// TIA Portal V16 export
// export: Created 2024-05-10T06:46:45.280441Z, ExportSetting WithDefaults, DisplayName Totally Integrated Automation Portal, DisplayVersion V16, DisplayName TIA Portal Version Control Interface, DisplayVersion V16, DisplayName TIA Portal Openness, DisplayVersion V16, DisplayName STEP 7 Professional, DisplayVersion V16, DisplayName STEP 7 Safety, DisplayVersion V16, DisplayName WinCC Professional, DisplayVersion V16
VAR_GLOBAL   // PLC tag table "105阀控制变量表"
   EN_阻挡下指令自动 AT %M2000.0 : Bool;
   EN_阻挡上指令自动 AT %M2000.1 : Bool;
   EN_提升机下指令自动 AT %M2000.4 : Bool;
   EN_提升机上指令自动 AT %M2000.5 : Bool;
   EX_阻挡下指令自动 AT %M2001.0 : Bool;
   EX_阻挡上指令自动 AT %M2001.1 : Bool;
   EX_提升机下指令自动 AT %M2001.4 : Bool;
   EX_提升机上指令自动 AT %M2001.5 : Bool;
   ST01上阻挡下指令自动 AT %M2002.0 : Bool;
   ST01上阻挡上指令自动 AT %M2002.1 : Bool;
   ST01下阻挡下指令自动 AT %M2002.4 : Bool;
   ST01下阻挡上指令自动 AT %M2002.5 : Bool;
   ST02上阻挡下指令自动 AT %M2003.0 : Bool;
   ST02上阻挡上指令自动 AT %M2003.1 : Bool;
   ST02下阻挡下指令自动 AT %M2003.4 : Bool;
   ST02下阻挡上指令自动 AT %M2003.5 : Bool;
   ST03上阻挡下指令自动 AT %M2004.0 : Bool;
   ST03上阻挡上指令自动 AT %M2004.1 : Bool;
   ST03下阻挡下指令自动 AT %M2004.4 : Bool;
   ST03下阻挡上指令自动 AT %M2004.5 : Bool;
   ST04上阻挡下指令自动 AT %M2005.0 : Bool;
   ST04上阻挡上指令自动 AT %M2005.1 : Bool;
   ST05上阻挡下指令自动 AT %M2005.4 : Bool;
   ST05上阻挡上指令自动 AT %M2005.5 : Bool;
   ST06上阻挡下指令自动 AT %M2006.0 : Bool;
   ST06上阻挡上指令自动 AT %M2006.1 : Bool;
   ST07上阻挡下指令自动 AT %M2006.4 : Bool;
   ST07上阻挡上指令自动 AT %M2006.5 : Bool;
   ST08上阻挡下指令自动 AT %M2007.0 : Bool;
   ST08上阻挡上指令自动 AT %M2007.1 : Bool;
   ST09上阻挡下指令自动 AT %M2007.4 : Bool;
   ST09上阻挡上指令自动 AT %M2007.5 : Bool;
   ST10上阻挡下指令自动 AT %M2008.0 : Bool;
   ST10上阻挡上指令自动 AT %M2008.1 : Bool;
   ST11上阻挡下指令自动 AT %M2008.4 : Bool;
   ST11上阻挡上指令自动 AT %M2008.5 : Bool;
   ST12上阻挡下指令自动 AT %M2009.0 : Bool;
   ST12上阻挡上指令自动 AT %M2009.1 : Bool;
   阀20进指令自动 AT %M2009.4 : Bool;
   阀20回指令自动 AT %M2009.5 : Bool;
   阀21进指令自动 AT %M2010.0 : Bool;
   阀21回指令自动 AT %M2010.1 : Bool;
   阀22进指令自动 AT %M2010.4 : Bool;
   阀22回指令自动 AT %M2010.5 : Bool;
   阀23进指令自动 AT %M2011.0 : Bool;
   阀23回指令自动 AT %M2011.1 : Bool;
   阀24进指令自动 AT %M2011.4 : Bool;
   阀24回指令自动 AT %M2011.5 : Bool;
   阀25进指令自动 AT %M2012.0 : Bool;
   阀25回指令自动 AT %M2012.1 : Bool;
   阀26进指令自动 AT %M2012.4 : Bool;
   阀26回指令自动 AT %M2012.5 : Bool;
   阀27进指令自动 AT %M2013.0 : Bool;
   阀27回指令自动 AT %M2013.1 : Bool;
   阀28进指令自动 AT %M2013.4 : Bool;
   阀28回指令自动 AT %M2013.5 : Bool;
   阀29进指令自动 AT %M2014.0 : Bool;
   阀29回指令自动 AT %M2014.1 : Bool;
   阀30进指令自动 AT %M2014.4 : Bool;
   阀30回指令自动 AT %M2014.5 : Bool;
   阀31进指令自动 AT %M2015.0 : Bool;
   阀31回指令自动 AT %M2015.1 : Bool;
   阀32进指令自动 AT %M2015.4 : Bool;
   阀32回指令自动 AT %M2015.5 : Bool;
   阀33进指令自动 AT %M2016.0 : Bool;
   阀33回指令自动 AT %M2016.1 : Bool;
   阀34进指令自动 AT %M2016.4 : Bool;
   阀34回指令自动 AT %M2016.5 : Bool;
   阀35进指令自动 AT %M2017.0 : Bool;
   阀35回指令自动 AT %M2017.1 : Bool;
   阀36进指令自动 AT %M2017.4 : Bool;
   阀36回指令自动 AT %M2017.5 : Bool;
   阀37进指令自动 AT %M2018.0 : Bool;
   阀37回指令自动 AT %M2018.1 : Bool;
   阀38进指令自动 AT %M2018.4 : Bool;
   阀38回指令自动 AT %M2018.5 : Bool;
   阀39进指令自动 AT %M2019.0 : Bool;
   阀39回指令自动 AT %M2019.1 : Bool;
   阀40进指令自动 AT %M2019.4 : Bool;
   阀40回指令自动 AT %M2019.5 : Bool;
   阀41进指令自动 AT %M2020.0 : Bool;
   阀41回指令自动 AT %M2020.1 : Bool;
   阀42进指令自动 AT %M2020.4 : Bool;
   阀42回指令自动 AT %M2020.5 : Bool;
   阀43进指令自动 AT %M2021.0 : Bool;
   阀43回指令自动 AT %M2021.1 : Bool;
   阀44进指令自动 AT %M2021.4 : Bool;
   阀44回指令自动 AT %M2021.5 : Bool;
   阀45进指令自动 AT %M2022.0 : Bool;
   阀45回指令自动 AT %M2022.1 : Bool;
   阀46进指令自动 AT %M2022.4 : Bool;
   阀46回指令自动 AT %M2022.5 : Bool;
   阀47进指令自动 AT %M2023.0 : Bool;
   阀47回指令自动 AT %M2023.1 : Bool;
   阀48进指令自动 AT %M2023.4 : Bool;
   阀48回指令自动 AT %M2023.5 : Bool;
   EN_阻挡下指令手动 AT %M1000.0 : Bool;
   EN_阻挡上指令手动 AT %M1000.1 : Bool;
   EN_提升机下指令手动 AT %M1000.4 : Bool;
   EN_提升机上指令手动 AT %M1000.5 : Bool;
   EX_阻挡下指令手动 AT %M1001.0 : Bool;
   EX_阻挡上指令手动 AT %M1001.1 : Bool;
   EX_提升机下指令手动 AT %M1001.4 : Bool;
   EX_提升机上指令手动 AT %M1001.5 : Bool;
   ST01上阻挡下指令手动 AT %M1002.0 : Bool;
   ST01上阻挡上指令手动 AT %M1002.1 : Bool;
   ST01下阻挡下指令手动 AT %M1002.4 : Bool;
   ST01下阻挡上指令手动 AT %M1002.5 : Bool;
   ST02上阻挡下指令手动 AT %M1003.0 : Bool;
   ST02上阻挡上指令手动 AT %M1003.1 : Bool;
   ST02下阻挡下指令手动 AT %M1003.4 : Bool;
   ST02下阻挡上指令手动 AT %M1003.5 : Bool;
   ST03上阻挡下指令手动 AT %M1004.0 : Bool;
   ST03上阻挡上指令手动 AT %M1004.1 : Bool;
   ST03下阻挡下指令手动 AT %M1004.4 : Bool;
   ST03下阻挡上指令手动 AT %M1004.5 : Bool;
   ST04上阻挡下指令手动 AT %M1005.0 : Bool;
   ST04上阻挡上指令手动 AT %M1005.1 : Bool;
   ST05上阻挡下指令手动 AT %M1005.4 : Bool;
   ST05上阻挡上指令手动 AT %M1005.5 : Bool;
   ST06上阻挡下指令手动 AT %M1006.0 : Bool;
   ST06上阻挡上指令手动 AT %M1006.1 : Bool;
   ST07上阻挡下指令手动 AT %M1006.4 : Bool;
   ST07上阻挡上指令手动 AT %M1006.5 : Bool;
   ST08上阻挡下指令手动 AT %M1007.0 : Bool;
   ST08上阻挡上指令手动 AT %M1007.1 : Bool;
   ST09上阻挡下指令手动 AT %M1007.4 : Bool;
   ST09上阻挡上指令手动 AT %M1007.5 : Bool;
   ST10上阻挡下指令手动 AT %M1008.0 : Bool;
   ST10上阻挡上指令手动 AT %M1008.1 : Bool;
   ST11上阻挡下指令手动 AT %M1008.4 : Bool;
   ST11上阻挡上指令手动 AT %M1008.5 : Bool;
   ST12上阻挡下指令手动 AT %M1009.0 : Bool;
   ST12上阻挡上指令手动 AT %M1009.1 : Bool;
   阀20进指令手动 AT %M1009.4 : Bool;
   阀20回指令手动 AT %M1009.5 : Bool;
   阀21进指令手动 AT %M1010.0 : Bool;
   阀21回指令手动 AT %M1010.1 : Bool;
   阀22进指令手动 AT %M1010.4 : Bool;
   阀22回指令手动 AT %M1010.5 : Bool;
   阀23进指令手动 AT %M1011.0 : Bool;
   阀23回指令手动 AT %M1011.1 : Bool;
   阀24进指令手动 AT %M1011.4 : Bool;
   阀24回指令手动 AT %M1011.5 : Bool;
   阀25进指令手动 AT %M1012.0 : Bool;
   阀25回指令手动 AT %M1012.1 : Bool;
   阀26进指令手动 AT %M1012.4 : Bool;
   阀26回指令手动 AT %M1012.5 : Bool;
   阀27进指令手动 AT %M1013.0 : Bool;
   阀27回指令手动 AT %M1013.1 : Bool;
   阀28进指令手动 AT %M1013.4 : Bool;
   阀28回指令手动 AT %M1013.5 : Bool;
   阀29进指令手动 AT %M1014.0 : Bool;
   阀29回指令手动 AT %M1014.1 : Bool;
   阀30进指令手动 AT %M1014.4 : Bool;
   阀30回指令手动 AT %M1014.5 : Bool;
   阀31进指令手动 AT %M1015.0 : Bool;
   阀31回指令手动 AT %M1015.1 : Bool;
   阀32进指令手动 AT %M1015.4 : Bool;
   阀32回指令手动 AT %M1015.5 : Bool;
   阀33进指令手动 AT %M1016.0 : Bool;
   阀33回指令手动 AT %M1016.1 : Bool;
   阀34进指令手动 AT %M1016.4 : Bool;
   阀34回指令手动 AT %M1016.5 : Bool;
   阀35进指令手动 AT %M1017.0 : Bool;
   阀35回指令手动 AT %M1017.1 : Bool;
   阀36进指令手动 AT %M1017.4 : Bool;
   阀36回指令手动 AT %M1017.5 : Bool;
   阀37进指令手动 AT %M1018.0 : Bool;
   阀37回指令手动 AT %M1018.1 : Bool;
   阀38进指令手动 AT %M1018.4 : Bool;
   阀38回指令手动 AT %M1018.5 : Bool;
   阀39进指令手动 AT %M1019.0 : Bool;
   阀39回指令手动 AT %M1019.1 : Bool;
   阀40进指令手动 AT %M1019.4 : Bool;
   阀40回指令手动 AT %M1019.5 : Bool;
   阀41进指令手动 AT %M1020.0 : Bool;
   阀41回指令手动 AT %M1020.1 : Bool;
   阀42进指令手动 AT %M1020.4 : Bool;
   阀42回指令手动 AT %M1020.5 : Bool;
   阀43进指令手动 AT %M1021.0 : Bool;
   阀43回指令手动 AT %M1021.1 : Bool;
   阀44进指令手动 AT %M1021.4 : Bool;
   阀44回指令手动 AT %M1021.5 : Bool;
   阀45进指令手动 AT %M1022.0 : Bool;
   阀45回指令手动 AT %M1022.1 : Bool;
   阀46进指令手动 AT %M1022.4 : Bool;
   阀46回指令手动 AT %M1022.5 : Bool;
   阀47进指令手动 AT %M1023.0 : Bool;
   阀47回指令手动 AT %M1023.1 : Bool;
   阀48进指令手动 AT %M1023.4 : Bool;
   阀48回指令手动 AT %M1023.5 : Bool;
   EN_阻挡下到位 AT %M3000.0 : Bool;
   EN_阻挡上到位 AT %M3000.1 : Bool;
   EN_提升机下到位 AT %M3000.4 : Bool;
   EN_提升机上到位 AT %M3000.5 : Bool;
   EX_阻挡下到位 AT %M3001.0 : Bool;
   EX_阻挡上到位 AT %M3001.1 : Bool;
   EX_提升机下到位 AT %M3001.4 : Bool;
   EX_提升机上到位 AT %M3001.5 : Bool;
   ST01上阻挡下到位 AT %M3002.0 : Bool;
   ST01上阻挡上到位 AT %M3002.1 : Bool;
   ST01下阻挡下到位 AT %M3002.4 : Bool;
   ST01下阻挡上到位 AT %M3002.5 : Bool;
   ST02上阻挡下到位 AT %M3003.0 : Bool;
   ST02上阻挡上到位 AT %M3003.1 : Bool;
   ST02下阻挡下到位 AT %M3003.4 : Bool;
   ST02下阻挡上到位 AT %M3003.5 : Bool;
   ST03上阻挡下到位 AT %M3004.0 : Bool;
   ST03上阻挡上到位 AT %M3004.1 : Bool;
   ST03下阻挡下到位 AT %M3004.4 : Bool;
   ST03下阻挡上到位 AT %M3004.5 : Bool;
   ST04上阻挡下到位 AT %M3005.0 : Bool;
   ST04上阻挡上到位 AT %M3005.1 : Bool;
   ST05上阻挡下到位 AT %M3005.4 : Bool;
   ST05上阻挡上到位 AT %M3005.5 : Bool;
   ST06上阻挡下到位 AT %M3006.0 : Bool;
   ST06上阻挡上到位 AT %M3006.1 : Bool;
   ST07上阻挡下到位 AT %M3006.4 : Bool;
   ST07上阻挡上到位 AT %M3006.5 : Bool;
   ST08上阻挡下到位 AT %M3007.0 : Bool;
   ST08上阻挡上到位 AT %M3007.1 : Bool;
   ST09上阻挡下到位 AT %M3007.4 : Bool;
   ST09上阻挡上到位 AT %M3007.5 : Bool;
   ST10上阻挡下到位 AT %M3008.0 : Bool;
   ST10上阻挡上到位 AT %M3008.1 : Bool;
   ST11上阻挡下到位 AT %M3008.4 : Bool;
   ST11上阻挡上到位 AT %M3008.5 : Bool;
   ST12上阻挡下到位 AT %M3009.0 : Bool;
   ST12上阻挡上到位 AT %M3009.1 : Bool;
   阀20进到位 AT %M3009.4 : Bool;
   阀20回到位 AT %M3009.5 : Bool;
   阀21进到位 AT %M3010.0 : Bool;
   阀21回到位 AT %M3010.1 : Bool;
   阀22进到位 AT %M3010.4 : Bool;
   阀22回到位 AT %M3010.5 : Bool;
   阀23进到位 AT %M3011.0 : Bool;
   阀23回到位 AT %M3011.1 : Bool;
   阀24进到位 AT %M3011.4 : Bool;
   阀24回到位 AT %M3011.5 : Bool;
   阀25进到位 AT %M3012.0 : Bool;
   阀25回到位 AT %M3012.1 : Bool;
   阀26进到位 AT %M3012.4 : Bool;
   阀26回到位 AT %M3012.5 : Bool;
   阀27进到位 AT %M3013.0 : Bool;
   阀27回到位 AT %M3013.1 : Bool;
   阀28进到位 AT %M3013.4 : Bool;
   阀28回到位 AT %M3013.5 : Bool;
   阀29进到位 AT %M3014.0 : Bool;
   阀29回到位 AT %M3014.1 : Bool;
   阀30进到位 AT %M3014.4 : Bool;
   阀30回到位 AT %M3014.5 : Bool;
   阀31进到位 AT %M3015.0 : Bool;
   阀31回到位 AT %M3015.1 : Bool;
   阀32进到位 AT %M3015.4 : Bool;
   阀32回到位 AT %M3015.5 : Bool;
   阀33进到位 AT %M3016.0 : Bool;
   阀33回到位 AT %M3016.1 : Bool;
   阀34进到位 AT %M3016.4 : Bool;
   阀34回到位 AT %M3016.5 : Bool;
   阀35进到位 AT %M3017.0 : Bool;
   阀35回到位 AT %M3017.1 : Bool;
   阀36进到位 AT %M3017.4 : Bool;
   阀36回到位 AT %M3017.5 : Bool;
   阀37进到位 AT %M3018.0 : Bool;
   阀37回到位 AT %M3018.1 : Bool;
   阀38进到位 AT %M3018.4 : Bool;
   阀38回到位 AT %M3018.5 : Bool;
   阀39进到位 AT %M3019.0 : Bool;
   阀39回到位 AT %M3019.1 : Bool;
   阀40进到位 AT %M3019.4 : Bool;
   阀40回到位 AT %M3019.5 : Bool;
   阀41进到位 AT %M3020.0 : Bool;
   阀41回到位 AT %M3020.1 : Bool;
   阀42进到位 AT %M3020.4 : Bool;
   阀42回到位 AT %M3020.5 : Bool;
   阀43进到位 AT %M3021.0 : Bool;
   阀43回到位 AT %M3021.1 : Bool;
   阀44进到位 AT %M3021.4 : Bool;
   阀44回到位 AT %M3021.5 : Bool;
   阀45进到位 AT %M3022.0 : Bool;
   阀45回到位 AT %M3022.1 : Bool;
   阀46进到位 AT %M3022.4 : Bool;
   阀46回到位 AT %M3022.5 : Bool;
   阀47进到位 AT %M3023.0 : Bool;
   阀47回到位 AT %M3023.1 : Bool;
   阀48进到位 AT %M3023.4 : Bool;
   阀48回到位 AT %M3023.5 : Bool;
   滚筒1正转指令自动 AT %M2100.0 : Bool;
   滚筒1反转指令自动 AT %M2100.1 : Bool;
   滚筒2正转指令自动 AT %M2100.4 : Bool;
   滚筒2反转指令自动 AT %M2100.5 : Bool;
   滚筒3正转指令自动 AT %M2101.0 : Bool;
   滚筒3反转指令自动 AT %M2101.1 : Bool;
   滚筒4正转指令自动 AT %M2101.4 : Bool;
   滚筒4反转指令自动 AT %M2101.5 : Bool;
   滚筒5正转指令自动 AT %M2102.0 : Bool;
   滚筒5反转指令自动 AT %M2102.1 : Bool;
   滚筒6正转指令自动 AT %M2102.4 : Bool;
   滚筒6反转指令自动 AT %M2102.5 : Bool;
   滚筒7正转指令自动 AT %M2103.0 : Bool;
   滚筒7反转指令自动 AT %M2103.1 : Bool;
   滚筒8正转指令自动 AT %M2103.4 : Bool;
   滚筒8反转指令自动 AT %M2103.5 : Bool;
   滚筒9正转指令自动 AT %M2104.0 : Bool;
   滚筒9反转指令自动 AT %M2104.1 : Bool;
   滚筒10正转指令自动 AT %M2104.4 : Bool;
   滚筒10反转指令自动 AT %M2104.5 : Bool;
   滚筒11正转指令自动 AT %M2105.0 : Bool;
   滚筒11反转指令自动 AT %M2105.1 : Bool;
   滚筒12正转指令自动 AT %M2105.4 : Bool;
   滚筒12反转指令自动 AT %M2105.5 : Bool;
   滚筒13正转指令自动 AT %M2106.0 : Bool;
   滚筒13反转指令自动 AT %M2106.1 : Bool;
   滚筒14正转指令自动 AT %M2106.4 : Bool;
   滚筒14反转指令自动 AT %M2106.5 : Bool;
   滚筒15正转指令自动 AT %M2107.0 : Bool;
   滚筒15反转指令自动 AT %M2107.1 : Bool;
   滚筒16正转指令自动 AT %M2107.4 : Bool;
   滚筒16反转指令自动 AT %M2107.5 : Bool;
   滚筒17正转指令自动 AT %M2108.0 : Bool;
   滚筒17反转指令自动 AT %M2108.1 : Bool;
   滚筒18正转指令自动 AT %M2108.4 : Bool;
   滚筒18反转指令自动 AT %M2108.5 : Bool;
   滚筒19正转指令自动 AT %M2109.0 : Bool;
   滚筒19反转指令自动 AT %M2109.1 : Bool;
   滚筒20正转指令自动 AT %M2109.4 : Bool;
   滚筒20反转指令自动 AT %M2109.5 : Bool;
   滚筒21正转指令自动 AT %M2110.0 : Bool;
   滚筒21反转指令自动 AT %M2110.1 : Bool;
   滚筒22正转指令自动 AT %M2110.4 : Bool;
   滚筒22反转指令自动 AT %M2110.5 : Bool;
   滚筒23正转指令自动 AT %M2111.0 : Bool;
   滚筒23反转指令自动 AT %M2111.1 : Bool;
   滚筒24正转指令自动 AT %M2111.4 : Bool;
   滚筒24反转指令自动 AT %M2111.5 : Bool;
   滚筒25正转指令自动 AT %M2112.0 : Bool;
   滚筒25反转指令自动 AT %M2112.1 : Bool;
   滚筒26正转指令自动 AT %M2112.4 : Bool;
   滚筒26反转指令自动 AT %M2112.5 : Bool;
   滚筒27正转指令自动 AT %M2113.0 : Bool;
   滚筒27反转指令自动 AT %M2113.1 : Bool;
   滚筒28正转指令自动 AT %M2113.4 : Bool;
   滚筒28反转指令自动 AT %M2113.5 : Bool;
   滚筒29正转指令自动 AT %M2114.0 : Bool;
   滚筒29反转指令自动 AT %M2114.1 : Bool;
   滚筒30正转指令自动 AT %M2114.4 : Bool;
   滚筒30反转指令自动 AT %M2114.5 : Bool;
   滚筒31正转指令自动 AT %M2115.0 : Bool;
   滚筒31反转指令自动 AT %M2115.1 : Bool;
   滚筒32正转指令自动 AT %M2115.4 : Bool;
   滚筒32反转指令自动 AT %M2115.5 : Bool;
   滚筒33正转指令自动 AT %M2116.0 : Bool;
   滚筒33反转指令自动 AT %M2116.1 : Bool;
   滚筒34正转指令自动 AT %M2116.4 : Bool;
   滚筒34反转指令自动 AT %M2116.5 : Bool;
   滚筒35正转指令自动 AT %M2117.0 : Bool;
   滚筒35反转指令自动 AT %M2117.1 : Bool;
   滚筒36正转指令自动 AT %M2117.4 : Bool;
   滚筒36反转指令自动 AT %M2117.5 : Bool;
   滚筒37正转指令自动 AT %M2118.0 : Bool;
   滚筒37反转指令自动 AT %M2118.1 : Bool;
   滚筒38正转指令自动 AT %M2118.4 : Bool;
   滚筒38反转指令自动 AT %M2118.5 : Bool;
   滚筒39正转指令自动 AT %M2119.0 : Bool;
   滚筒39反转指令自动 AT %M2119.1 : Bool;
   滚筒40正转指令自动 AT %M2119.4 : Bool;
   滚筒40反转指令自动 AT %M2119.5 : Bool;
   滚筒41正转指令自动 AT %M2120.0 : Bool;
   滚筒41反转指令自动 AT %M2120.1 : Bool;
   滚筒42正转指令自动 AT %M2120.4 : Bool;
   滚筒42反转指令自动 AT %M2120.5 : Bool;
   滚筒43正转指令自动 AT %M2121.0 : Bool;
   滚筒43反转指令自动 AT %M2121.1 : Bool;
   滚筒44正转指令自动 AT %M2121.4 : Bool;
   滚筒44反转指令自动 AT %M2121.5 : Bool;
   滚筒45正转指令自动 AT %M2122.0 : Bool;
   滚筒45反转指令自动 AT %M2122.1 : Bool;
   滚筒46正转指令自动 AT %M2122.4 : Bool;
   滚筒46反转指令自动 AT %M2122.5 : Bool;
   滚筒47正转指令自动 AT %M2123.0 : Bool;
   滚筒47反转指令自动 AT %M2123.1 : Bool;
   滚筒48正转指令自动 AT %M2123.4 : Bool;
   滚筒48反转指令自动 AT %M2123.5 : Bool;
   滚筒1正转指令手动 AT %M1100.0 : Bool;
   滚筒1反转指令手动 AT %M1100.1 : Bool;
   滚筒2正转指令手动 AT %M1100.4 : Bool;
   滚筒2反转指令手动 AT %M1100.5 : Bool;
   滚筒3正转指令手动 AT %M1101.0 : Bool;
   滚筒3反转指令手动 AT %M1101.1 : Bool;
   滚筒4正转指令手动 AT %M1101.4 : Bool;
   滚筒4反转指令手动 AT %M1101.5 : Bool;
   滚筒5正转指令手动 AT %M1102.0 : Bool;
   滚筒5反转指令手动 AT %M1102.1 : Bool;
   滚筒6正转指令手动 AT %M1102.4 : Bool;
   滚筒6反转指令手动 AT %M1102.5 : Bool;
   滚筒7正转指令手动 AT %M1103.0 : Bool;
   滚筒7反转指令手动 AT %M1103.1 : Bool;
   滚筒8正转指令手动 AT %M1103.4 : Bool;
   滚筒8反转指令手动 AT %M1103.5 : Bool;
   滚筒9正转指令手动 AT %M1104.0 : Bool;
   滚筒9反转指令手动 AT %M1104.1 : Bool;
   滚筒10正转指令手动 AT %M1104.4 : Bool;
   滚筒10反转指令手动 AT %M1104.5 : Bool;
   滚筒11正转指令手动 AT %M1105.0 : Bool;
   滚筒11反转指令手动 AT %M1105.1 : Bool;
   滚筒12正转指令手动 AT %M1105.4 : Bool;
   滚筒12反转指令手动 AT %M1105.5 : Bool;
   滚筒13正转指令手动 AT %M1106.0 : Bool;
   滚筒13反转指令手动 AT %M1106.1 : Bool;
   滚筒14正转指令手动 AT %M1106.4 : Bool;
   滚筒14反转指令手动 AT %M1106.5 : Bool;
   滚筒15正转指令手动 AT %M1107.0 : Bool;
   滚筒15反转指令手动 AT %M1107.1 : Bool;
   滚筒16正转指令手动 AT %M1107.4 : Bool;
   滚筒16反转指令手动 AT %M1107.5 : Bool;
   滚筒17正转指令手动 AT %M1108.0 : Bool;
   滚筒17反转指令手动 AT %M1108.1 : Bool;
   滚筒18正转指令手动 AT %M1108.4 : Bool;
   滚筒18反转指令手动 AT %M1108.5 : Bool;
   滚筒19正转指令手动 AT %M1109.0 : Bool;
   滚筒19反转指令手动 AT %M1109.1 : Bool;
   滚筒20正转指令手动 AT %M1109.4 : Bool;
   滚筒20反转指令手动 AT %M1109.5 : Bool;
   滚筒21正转指令手动 AT %M1110.0 : Bool;
   滚筒21反转指令手动 AT %M1110.1 : Bool;
   滚筒22正转指令手动 AT %M1110.4 : Bool;
   滚筒22反转指令手动 AT %M1110.5 : Bool;
   滚筒23正转指令手动 AT %M1111.0 : Bool;
   滚筒23反转指令手动 AT %M1111.1 : Bool;
   滚筒24正转指令手动 AT %M1111.4 : Bool;
   滚筒24反转指令手动 AT %M1111.5 : Bool;
   滚筒25正转指令手动 AT %M1112.0 : Bool;
   滚筒25反转指令手动 AT %M1112.1 : Bool;
   滚筒26正转指令手动 AT %M1112.4 : Bool;
   滚筒26反转指令手动 AT %M1112.5 : Bool;
   滚筒27正转指令手动 AT %M1113.0 : Bool;
   滚筒27反转指令手动 AT %M1113.1 : Bool;
   滚筒28正转指令手动 AT %M1113.4 : Bool;
   滚筒28反转指令手动 AT %M1113.5 : Bool;
   滚筒29正转指令手动 AT %M1114.0 : Bool;
   滚筒29反转指令手动 AT %M1114.1 : Bool;
   滚筒30正转指令手动 AT %M1114.4 : Bool;
   滚筒30反转指令手动 AT %M1114.5 : Bool;
   滚筒31正转指令手动 AT %M1115.0 : Bool;
   滚筒31反转指令手动 AT %M1115.1 : Bool;
   滚筒32正转指令手动 AT %M1115.4 : Bool;
   滚筒32反转指令手动 AT %M1115.5 : Bool;
   滚筒33正转指令手动 AT %M1116.0 : Bool;
   滚筒33反转指令手动 AT %M1116.1 : Bool;
   滚筒34正转指令手动 AT %M1116.4 : Bool;
   滚筒34反转指令手动 AT %M1116.5 : Bool;
   滚筒35正转指令手动 AT %M1117.0 : Bool;
   滚筒35反转指令手动 AT %M1117.1 : Bool;
   滚筒36正转指令手动 AT %M1117.4 : Bool;
   滚筒36反转指令手动 AT %M1117.5 : Bool;
   滚筒37正转指令手动 AT %M1118.0 : Bool;
   滚筒37反转指令手动 AT %M1118.1 : Bool;
   滚筒38正转指令手动 AT %M1118.4 : Bool;
   滚筒38反转指令手动 AT %M1118.5 : Bool;
   滚筒39正转指令手动 AT %M1119.0 : Bool;
   滚筒39反转指令手动 AT %M1119.1 : Bool;
   滚筒40正转指令手动 AT %M1119.4 : Bool;
   滚筒40反转指令手动 AT %M1119.5 : Bool;
   滚筒41正转指令手动 AT %M1120.0 : Bool;
   滚筒41反转指令手动 AT %M1120.1 : Bool;
   滚筒42正转指令手动 AT %M1120.4 : Bool;
   滚筒42反转指令手动 AT %M1120.5 : Bool;
   滚筒43正转指令手动 AT %M1121.0 : Bool;
   滚筒43反转指令手动 AT %M1121.1 : Bool;
   滚筒44正转指令手动 AT %M1121.4 : Bool;
   滚筒44反转指令手动 AT %M1121.5 : Bool;
   滚筒45正转指令手动 AT %M1122.0 : Bool;
   滚筒45反转指令手动 AT %M1122.1 : Bool;
   滚筒46正转指令手动 AT %M1122.4 : Bool;
   滚筒46反转指令手动 AT %M1122.5 : Bool;
   滚筒47正转指令手动 AT %M1123.0 : Bool;
   滚筒47反转指令手动 AT %M1123.1 : Bool;
   滚筒48正转指令手动 AT %M1123.4 : Bool;
   滚筒48反转指令手动 AT %M1123.5 : Bool;
   "滚筒1正转到位(不用" AT %M3100.0 : Bool;
   "滚筒1反转到位(不用" AT %M3100.1 : Bool;
   "滚筒2正转到位(不用" AT %M3100.4 : Bool;
   "滚筒2反转到位(不用" AT %M3100.5 : Bool;
   "滚筒3正转到位(不用" AT %M3101.0 : Bool;
   "滚筒3反转到位(不用" AT %M3101.1 : Bool;
   "滚筒4正转到位(不用" AT %M3101.4 : Bool;
   "滚筒4反转到位(不用" AT %M3101.5 : Bool;
   "滚筒5正转到位(不用" AT %M3102.0 : Bool;
   "滚筒5反转到位(不用" AT %M3102.1 : Bool;
   "滚筒6正转到位(不用" AT %M3102.4 : Bool;
   "滚筒6反转到位(不用" AT %M3102.5 : Bool;
   "滚筒7正转到位(不用" AT %M3103.0 : Bool;
   "滚筒7反转到位(不用" AT %M3103.1 : Bool;
   "滚筒8正转到位(不用" AT %M3103.4 : Bool;
   "滚筒8反转到位(不用" AT %M3103.5 : Bool;
   "滚筒9正转到位(不用" AT %M3104.0 : Bool;
   "滚筒9反转到位(不用" AT %M3104.1 : Bool;
   "滚筒10正转到位(不用" AT %M3104.4 : Bool;
   "滚筒10反转到位(不用" AT %M3104.5 : Bool;
   "滚筒11正转到位(不用" AT %M3105.0 : Bool;
   "滚筒11反转到位(不用" AT %M3105.1 : Bool;
   "滚筒12正转到位(不用" AT %M3105.4 : Bool;
   "滚筒12反转到位(不用" AT %M3105.5 : Bool;
   "滚筒13正转到位(不用" AT %M3106.0 : Bool;
   "滚筒13反转到位(不用" AT %M3106.1 : Bool;
   "滚筒14正转到位(不用" AT %M3106.4 : Bool;
   "滚筒14反转到位(不用" AT %M3106.5 : Bool;
   "滚筒15正转到位(不用" AT %M3107.0 : Bool;
   "滚筒15反转到位(不用" AT %M3107.1 : Bool;
   "滚筒16正转到位(不用" AT %M3107.4 : Bool;
   "滚筒16反转到位(不用" AT %M3107.5 : Bool;
   "滚筒17正转到位(不用" AT %M3108.0 : Bool;
   "滚筒17反转到位(不用" AT %M3108.1 : Bool;
   "滚筒18正转到位(不用" AT %M3108.4 : Bool;
   "滚筒18反转到位(不用" AT %M3108.5 : Bool;
   "滚筒19正转到位(不用" AT %M3109.0 : Bool;
   "滚筒19反转到位(不用" AT %M3109.1 : Bool;
   "滚筒20正转到位(不用" AT %M3109.4 : Bool;
   "滚筒20反转到位(不用" AT %M3109.5 : Bool;
   "滚筒21正转到位(不用" AT %M3110.0 : Bool;
   "滚筒21反转到位(不用" AT %M3110.1 : Bool;
   "滚筒22正转到位(不用" AT %M3110.4 : Bool;
   "滚筒22反转到位(不用" AT %M3110.5 : Bool;
   "滚筒23正转到位(不用" AT %M3111.0 : Bool;
   "滚筒23反转到位(不用" AT %M3111.1 : Bool;
   "滚筒24正转到位(不用" AT %M3111.4 : Bool;
   "滚筒24反转到位(不用" AT %M3111.5 : Bool;
   "滚筒25正转到位(不用" AT %M3112.0 : Bool;
   "滚筒25反转到位(不用" AT %M3112.1 : Bool;
   "滚筒26正转到位(不用" AT %M3112.4 : Bool;
   "滚筒26反转到位(不用" AT %M3112.5 : Bool;
   "滚筒27正转到位(不用" AT %M3113.0 : Bool;
   "滚筒27反转到位(不用" AT %M3113.1 : Bool;
   "滚筒28正转到位(不用" AT %M3113.4 : Bool;
   "滚筒28反转到位(不用" AT %M3113.5 : Bool;
   "滚筒29正转到位(不用" AT %M3114.0 : Bool;
   "滚筒29反转到位(不用" AT %M3114.1 : Bool;
   "滚筒30正转到位(不用" AT %M3114.4 : Bool;
   "滚筒30反转到位(不用" AT %M3114.5 : Bool;
   "滚筒31正转到位(不用" AT %M3115.0 : Bool;
   "滚筒31反转到位(不用" AT %M3115.1 : Bool;
   "滚筒32正转到位(不用" AT %M3115.4 : Bool;
   "滚筒32反转到位(不用" AT %M3115.5 : Bool;
   "滚筒33正转到位(不用" AT %M3116.0 : Bool;
   "滚筒33反转到位(不用" AT %M3116.1 : Bool;
   "滚筒34正转到位(不用" AT %M3116.4 : Bool;
   "滚筒34反转到位(不用" AT %M3116.5 : Bool;
   "滚筒35正转到位(不用" AT %M3117.0 : Bool;
   "滚筒35反转到位(不用" AT %M3117.1 : Bool;
   "滚筒36正转到位(不用" AT %M3117.4 : Bool;
   "滚筒36反转到位(不用" AT %M3117.5 : Bool;
   "滚筒37正转到位(不用" AT %M3118.0 : Bool;
   "滚筒37反转到位(不用" AT %M3118.1 : Bool;
   "滚筒38正转到位(不用" AT %M3118.4 : Bool;
   "滚筒38反转到位(不用" AT %M3118.5 : Bool;
   "滚筒39正转到位(不用" AT %M3119.0 : Bool;
   "滚筒39反转到位(不用" AT %M3119.1 : Bool;
   "滚筒40正转到位(不用" AT %M3119.4 : Bool;
   "滚筒40反转到位(不用" AT %M3119.5 : Bool;
   "滚筒41正转到位(不用" AT %M3120.0 : Bool;
   "滚筒41反转到位(不用" AT %M3120.1 : Bool;
   "滚筒42正转到位(不用" AT %M3120.4 : Bool;
   "滚筒42反转到位(不用" AT %M3120.5 : Bool;
   "滚筒43正转到位(不用" AT %M3121.0 : Bool;
   "滚筒43反转到位(不用" AT %M3121.1 : Bool;
   "滚筒44正转到位(不用" AT %M3121.4 : Bool;
   "滚筒44反转到位(不用" AT %M3121.5 : Bool;
   "滚筒45正转到位(不用" AT %M3122.0 : Bool;
   "滚筒45反转到位(不用" AT %M3122.1 : Bool;
   "滚筒46正转到位(不用" AT %M3122.4 : Bool;
   "滚筒46反转到位(不用" AT %M3122.5 : Bool;
   "滚筒47正转到位(不用" AT %M3123.0 : Bool;
   "滚筒47反转到位(不用" AT %M3123.1 : Bool;
   "滚筒48正转到位(不用" AT %M3123.4 : Bool;
   "滚筒48反转到位(不用" AT %M3123.5 : Bool;
   变频器1正转指令自动 AT %M2200.0 : Bool;
   变频器1反转指令自动 AT %M2200.1 : Bool;
   变频器2正转指令自动 AT %M2200.4 : Bool;
   变频器2反转指令自动 AT %M2200.5 : Bool;
   变频器3正转指令自动 AT %M2201.0 : Bool;
   变频器3反转指令自动 AT %M2201.1 : Bool;
   变频器4正转指令自动 AT %M2201.4 : Bool;
   变频器4反转指令自动 AT %M2201.5 : Bool;
   变频器5正转指令自动 AT %M2202.0 : Bool;
   变频器5反转指令自动 AT %M2202.1 : Bool;
   变频器6正转指令自动 AT %M2202.4 : Bool;
   变频器6反转指令自动 AT %M2202.5 : Bool;
   变频器7正转指令自动 AT %M2203.0 : Bool;
   变频器7反转指令自动 AT %M2203.1 : Bool;
   变频器8正转指令自动 AT %M2203.4 : Bool;
   变频器8反转指令自动 AT %M2203.5 : Bool;
   变频器9正转指令自动 AT %M2204.0 : Bool;
   变频器9反转指令自动 AT %M2204.1 : Bool;
   变频器10正转指令自动 AT %M2204.4 : Bool;
   变频器10反转指令自动 AT %M2204.5 : Bool;
   变频器11正转指令自动 AT %M2205.0 : Bool;
   变频器11反转指令自动 AT %M2205.1 : Bool;
   变频器12正转指令自动 AT %M2205.4 : Bool;
   变频器12反转指令自动 AT %M2205.5 : Bool;
   变频器13正转指令自动 AT %M2206.0 : Bool;
   变频器13反转指令自动 AT %M2206.1 : Bool;
   变频器14正转指令自动 AT %M2206.4 : Bool;
   变频器14反转指令自动 AT %M2206.5 : Bool;
   变频器15正转指令自动 AT %M2207.0 : Bool;
   变频器15反转指令自动 AT %M2207.1 : Bool;
   变频器16正转指令自动 AT %M2207.4 : Bool;
   变频器16反转指令自动 AT %M2207.5 : Bool;
   变频器1正转指令手动 AT %M1200.0 : Bool;
   变频器1反转指令手动 AT %M1200.1 : Bool;
   变频器2正转指令手动 AT %M1200.4 : Bool;
   变频器2反转指令手动 AT %M1200.5 : Bool;
   变频器3正转指令手动 AT %M1201.0 : Bool;
   变频器3反转指令手动 AT %M1201.1 : Bool;
   变频器4正转指令手动 AT %M1201.4 : Bool;
   变频器4反转指令手动 AT %M1201.5 : Bool;
   变频器5正转指令手动 AT %M1202.0 : Bool;
   变频器5反转指令手动 AT %M1202.1 : Bool;
   变频器6正转指令手动 AT %M1202.4 : Bool;
   变频器6反转指令手动 AT %M1202.5 : Bool;
   变频器7正转指令手动 AT %M1203.0 : Bool;
   变频器7反转指令手动 AT %M1203.1 : Bool;
   变频器8正转指令手动 AT %M1203.4 : Bool;
   变频器8反转指令手动 AT %M1203.5 : Bool;
   变频器9正转指令手动 AT %M1204.0 : Bool;
   变频器9反转指令手动 AT %M1204.1 : Bool;
   变频器10正转指令手动 AT %M1204.4 : Bool;
   变频器10反转指令手动 AT %M1204.5 : Bool;
   变频器11正转指令手动 AT %M1205.0 : Bool;
   变频器11反转指令手动 AT %M1205.1 : Bool;
   变频器12正转指令手动 AT %M1205.4 : Bool;
   变频器12反转指令手动 AT %M1205.5 : Bool;
   变频器13正转指令手动 AT %M1206.0 : Bool;
   变频器13反转指令手动 AT %M1206.1 : Bool;
   变频器14正转指令手动 AT %M1206.4 : Bool;
   变频器14反转指令手动 AT %M1206.5 : Bool;
   变频器15正转指令手动 AT %M1207.0 : Bool;
   变频器15反转指令手动 AT %M1207.1 : Bool;
   变频器16正转指令手动 AT %M1207.4 : Bool;
   变频器16反转指令手动 AT %M1207.5 : Bool;
   "变频器1正转到位(不用" AT %M3200.0 : Bool;
   "变频器1反转到位(不用" AT %M3200.1 : Bool;
   "变频器2正转到位(不用" AT %M3200.4 : Bool;
   "变频器2反转到位(不用" AT %M3200.5 : Bool;
   "变频器3正转到位(不用" AT %M3201.0 : Bool;
   "变频器3反转到位(不用" AT %M3201.1 : Bool;
   "变频器4正转到位(不用" AT %M3201.4 : Bool;
   "变频器4反转到位(不用" AT %M3201.5 : Bool;
   "变频器5正转到位(不用" AT %M3202.0 : Bool;
   "变频器5反转到位(不用" AT %M3202.1 : Bool;
   "变频器6正转到位(不用" AT %M3202.4 : Bool;
   "变频器6反转到位(不用" AT %M3202.5 : Bool;
   "变频器7正转到位(不用" AT %M3203.0 : Bool;
   "变频器7反转到位(不用" AT %M3203.1 : Bool;
   "变频器8正转到位(不用" AT %M3203.4 : Bool;
   "变频器8反转到位(不用" AT %M3203.5 : Bool;
   "变频器9正转到位(不用" AT %M3204.0 : Bool;
   "变频器9反转到位(不用" AT %M3204.1 : Bool;
   "变频器10正转到位(不用" AT %M3204.4 : Bool;
   "变频器10反转到位(不用" AT %M3204.5 : Bool;
   "变频器11正转到位(不用" AT %M3205.0 : Bool;
   "变频器11反转到位(不用" AT %M3205.1 : Bool;
   "变频器12正转到位(不用" AT %M3205.4 : Bool;
   "变频器12反转到位(不用" AT %M3205.5 : Bool;
   "变频器13正转到位(不用" AT %M3206.0 : Bool;
   "变频器13反转到位(不用" AT %M3206.1 : Bool;
   "变频器14正转到位(不用" AT %M3206.4 : Bool;
   "变频器14反转到位(不用" AT %M3206.5 : Bool;
   "变频器15正转到位(不用" AT %M3207.0 : Bool;
   "变频器15反转到位(不用" AT %M3207.1 : Bool;
   "变频器16正转到位(不用" AT %M3207.4 : Bool;
   "变频器16反转到位(不用" AT %M3207.5 : Bool;
END_VAR
